// TIA Portal V20 export
DATA_BLOCK "HmiInterface"   // DB45
// stored: Access Published, MemoryReserve 100, Namespace Unit1.Em5
   VAR
      em : "LAF_typeEmInterface";
      cm : "Unit1.Em5.typeCmHmiInterface";
      transferPnPLeft : "LER_typeSequenceInterface";
      transferPnPRight : "LER_typeSequenceInterface";
      GRnR_TransferPnP : "LER_typeSequenceInterface";
      cmTransferPnPLeftSafetyPin : "LBC_typeDigitalSignalInterface";
      cmTransferPnPLeftJRDetect : "LBC_typeDigitalSignalInterface";
      cmTransferPnPRightSafetyPin : "LBC_typeDigitalSignalInterface";
      cmTransferPnPRightJRDetect : "LBC_typeDigitalSignalInterface";
   END_VAR
   VAR RETAIN
      cmTransferPnPLeftAxisX : "LBC_typeAxis64PosInterface";
      cmTransferPnPLeftAxisY : "LBC_typeAxis64PosInterface";
      cmTransferPnPLeftAxisZ : "LBC_typeAxis64PosInterface";
      cmTransferPnPRightAxisX : "LBC_typeAxis64PosInterface";
      cmTransferPnPRightAxisY : "LBC_typeAxis64PosInterface";
      cmTransferPnPRightAxisZ : "LBC_typeAxis64PosInterface";
   END_VAR
   VAR
      cmTransferPnPLeftClampOpenClose : "LBC_typeTwoWayActuatorInterface";
      cmTransferPnPRightClampOpenClose : "LBC_typeTwoWayActuatorInterface";
      intCondition : "Unit1.Em5.typeIntConditionHmiInterface";
   END_VAR
BEGIN
   cmTransferPnPLeftAxisX.configuration.setPositions[0]."name" := 'Wait';
   cmTransferPnPLeftAxisX.configuration.setPositions[1]."name" := 'Side Tape';
   cmTransferPnPLeftAxisX.configuration.setPositions[2]."name" := 'Hot Press Left';
   cmTransferPnPLeftAxisX.configuration.setPositions[3]."name" := 'Hot Press Right';
   cmTransferPnPLeftAxisX.configuration.setPositions[4]."name" := 'Hipot & Thickness';
   cmTransferPnPLeftAxisX.configuration.setPositions[9]."name" := 'Side Tape Zone';
END_DATA_BLOCK
